TEXTLIST TextList_SettingPage_2
  1 = 'STATION 01'
  2 = 'STATION 02'
  3 = 'STATION 03'
  4 = 'STATION 04'
  5 = 'STATION 05'
  6 = 'STATION 06'
  7 = 'LOADING'
  8 = 'UNLOADING'
  9 = 'GENERAL'
   = ''
END_TEXTLIST

(* stored: Version 1.1.0.1, ProductVersion 3.1.4024.12
   TextList TextList_SettingPage_2: Id {02f2290c-8ea8-4e70-999e-c4e3abfd17ba} *)
